(* CoDeSys 2.3 export: ST_JALOUSIE.EXP *)

(* Data type *)
TYPE ST_Jalousie :
STRUCT
	mTimestruct: TIMESTRUCT;
	mPos: BYTE;

	mFbJalousie: FB_Jalousie;
END_STRUCT
END_TYPE
